(* PLC project CoDeSys External Library Template, WAGO e!COCKPIT e!COCKPIT, author 3S - Smart Software Solutions GmbH *)
(* stored: creationDateTime 2019-10-29T12:22:40.7625589, version 3.5.5.30, modificationDateTime 2019-10-24T14:40:07.960949, organization 3S - Smart Software Solutions GmbH *)
(* Library project template with all possible element types, docu and a sample project structure *)

FUNCTION_BLOCK fbUDPComm
  VAR_INPUT
    sIDSterownika : STRING;  (* ID sterownika *)
    sIDAplikacji : STRING;  (* ID aplikacji *)
    sMnemonik : STRING;  (* mnemonik właściciela *)
    sMACAdres : STRING;  (* MAC adres urządzenia - alias *)
    sMACAdresAplikacji : STRING;  (* MAC adres aplikacji - alias *)
    abMACAdresAplikacji : ARRAY[1..6] OF BYTE;  (* MAC adres aplikacji - wartość rzeczywista *)
    sDaneZapasowe : STRING;  (* dane zapasowe *)
    sAdresIP : STRING;  (* adres IP aplikacji *)
    wTransmitterPort : WORD;  (* port do wysyłania komunikatów *)
    wReceiverPort : WORD;  (* port nasłuchu *)
    sKluczSzyfrowania : STRING;
    intTablicaKomunikatowRozmiar : INT;
    intTablicaKomunikatowOverflow : INT;
    intTablicaKomunikatowZnacznikOdczytu : INT;
    iDetekcjaBlokadaKomunikacjiLimitIlosciRamek : INT;  (* Limit ilosi ramek do wysłania *)
    tDetekcjaBlokadaKomunikacjiLimitCzasu : TIME;
  END_VAR
  VAR_IN_OUT
    arTablicaKomunikatow : alARRAYTablicaKomunikatow;
    intTablicaKomunikatowZnacznikZapisu : INT;
    intTablicaKomunikatowZnacznikWysylkiUDP : INT;
    intTablicaKomunikatowLiczbaWBuforze : INT;
    intTransmitterLicznikKomunikatowWyslanych : INT;  (* zmienna zwierająca licznik komunikatów wysłanych pomiędzy heartbetami *)
    intReceiverLicznikKomunikatowOtrzymanych : INT;  (* zmienna zwierająca licznik komunikatów otrzymanych pomiędzy heartbetami *)
  END_VAR
  VAR
    fbTransmitter : fbBroadcaster;  (* definicja drivera wysyłającego broadcast pakietów UDP *)
    udiTransmitterNBytes : UDINT;  (* parametr drivera - ilość bajtów do wysłania *)
    xTransmitterClose : BOOL;  (* parametr drivera - zamknięcie portu komunikacyjnego *)
    xTransmitterTrigger : BOOL;  (* parametr drivera - uruchomienie wysłania telegramu *)
    sTransmitterTelegram : alSTRINGKomunikat;  (* zmienna zawierająca telegram do wysłania *)
    arTransmitterBuffer : ARRAY[1..512] OF BYTE;  (* tablica WORD bufora wysyłkowego *)
    pTransmitterBuffer : POINTER TO BYTE := ADR(arTransmitterBuffer[1]);  (* parametr drivera - pointer do tablicy bufora dla drivera wysyłającego *)
    fbReceiver : fbUdpReceiver;  (* definicja drivera odbierającego pakiety UDP *)
    xReceiverEnable : BOOL := TRUE;  (* parametr drivera - aktywacja działania drivera *)
    xReceiverOpen : BOOL := TRUE;  (* parametr drivera - otworzenie portu komunikacyjnego *)
    sReceiverTelegram : alSTRINGKomunikat;  (* zmienna zawierająca odebrany telegram *)
    arReceiverBuffer : ARRAY[1..512] OF BYTE;
    pReceiverBuffer : POINTER TO BYTE := ADR(arReceiverBuffer[1]);  (* parametr drivera - pointer do tablicy bufora dla drivera odbierającego *)
    intPetla : INT;  (* zmienna tymczasowa używana dla pętli *)
    arwHeartbeatTelegram : ARRAY[1..512] OF WORD;
    negUdpCommTxDone : F_TRIG;
    wCRC16_standard : WORD;
    intBlad : INT;
    sDane : alSTRINGKomunikat;
    sWyslanyKomunikat : alSTRINGKomunikat;
    typKomunikat : typKomunikat;
    xCRC16PakietOdebranyPoprawny : BOOL;
    arErrorKomunikat : ARRAY[0..20] OF alSTRINGKomunikat;  (* tablica przechowująca ostatni komunikat alarmu z danego kodu *)
    arErrorStan : ARRAY[1..20] OF BOOL;  (* tablica przechowująca stany alarmowe *)
    intTabelaKomunikatowZnacznikOdczytu : INT := 1;
    intEmergencyStopActiveZaraportowana : INT;
    sWyslanyKomunikatDummy : STRING;
    BlokadaKomunikacjiDetekcjaTriger : RS;  (* Blokada wysylania komunikatów *)
    BlokadaKomunikacjiDetekcjaTimer : TON;
    BlokadaKomunikacjiTriger : RS;
    fbBlokadaKomunikacjiTimer : TON;  (* Timer do cyklicznego wysyłania ramki z errorem blokady wysyłania ramek *)
    xBlokadaKomunikacji : BOOL;  (* Blokada komunikacji *)
    BlokadaKomunikacjiTimeDiff : TIME := TIME#200m0s0ms;
    xWyslijErrorBlokadyKomunikacji : BOOL;  (* Zmienna pomocniczna do fbWyslijErrorBlokadyKomunikacji *)
    fbWyslijErrorBlokadyKomunikacji : F_TRIG;  (* Zbocze opadające xWyslijErrorBlokadyKomunikacji *)
    xBlokadaKomunikacjiReset : BOOL;  (* Reset blokady komunikacji *)
    timestamp : STRING;  (* obsługa debugowania problemów z komunikatami *)
    dtCzasLokalny : DT;
    dtCzasKomunikatu : DT;
    tPrzesuniecie : TIME := TIME#5m0s0ms;
    xPrzekroczony : BOOL := FALSE;
    arTablicaBlednychKomunikatow : alARRAYTablicaKomunikatowDebug;
    uintZnacznikTablicyBlednychKomunikatow : UINT := 1;
    intTablicaKomunikatowZnacznikWysylkiUDP_Pamiec : INT := -1;
  END_VAR

            // jeśli wysyłanie telegramu zakończone OK wyczyść zmienną zawierającą telegram oraz wyzeruj licznik komunikatów wysłanych jeśli TO BYł heartbeat
// 2019-04-01 - JC Dodanie blokady wysylania komunikatów w przypadku przekroczenia limitu
// 2019-04-18 - AWy: Wysyłanie ramki z errorem blokady wysyłania ramek co minutę
// 2019-04-19 - AWy: Poprawienie mechanizmu resetu blokady i usunięcie tBlokadaKomunikacjiOpoznienie
// 2019-04-25 - AWy: Przeniesienie xBlokadaKomunikacjiReset z VAR_INPUT do VAR
// 2019-10-24 - AWy: Zmiana tPrzesuniecie na 300 sekund
IF NOT xTransmitterTrigger AND sTransmitterTelegram <> '' THEN
	IF fnKomunikatTyp(sTransmitterTelegram) = 'H' THEN
		intTransmitterLicznikKomunikatowWyslanych := 0;
	END_IF
	sTransmitterTelegram := '';
END_IF

IF sTransmitterTelegram = '' AND intTablicaKomunikatowZnacznikWysylkiUDP <> intTablicaKomunikatowZnacznikZapisu THEN
	fnTablicaKomunikatowInkrementacja(intWskaznik := intTablicaKomunikatowZnacznikWysylkiUDP , intRozmiarTablicy := intTablicaKomunikatowRozmiar);
	WHILE fnKomunikatMACAdres(arTablicaKomunikatow[intTablicaKomunikatowZnacznikWysylkiUDP]) <> sMACAdres AND intTablicaKomunikatowZnacznikWysylkiUDP <> intTablicaKomunikatowZnacznikZapisu DO
		fnTablicaKomunikatowInkrementacja(intWskaznik := intTablicaKomunikatowZnacznikWysylkiUDP , intRozmiarTablicy := intTablicaKomunikatowRozmiar);
 	END_WHILE
	IF fnKomunikatMACAdres(arTablicaKomunikatow[intTablicaKomunikatowZnacznikWysylkiUDP]) = sMACAdres THEN
		intTransmitterLicznikKomunikatowWyslanych := intTransmitterLicznikKomunikatowWyslanych + 1;
		//////////////////////////////////
		//Walidacja poprawności komunikatu
		//////////////////////////////////
		IF intTablicaKomunikatowZnacznikWysylkiUDP_Pamiec <> intTablicaKomunikatowZnacznikWysylkiUDP THEN
			timestamp := fnKomunikatSprawdzTimeStamp( sKomunikat:= arTablicaKomunikatow[intTablicaKomunikatowZnacznikWysylkiUDP],dtDataCzasWKomunikacie:=dtCzasKomunikatu, dtDataCzasAktualny:=dtCzasLokalny);
			IF(dtCzasKomunikatu + tPrzesuniecie) < dtCzasLokalny THEN
				xPrzekroczony := TRUE;
				arTablicaBlednychKomunikatow[uintZnacznikTablicyBlednychKomunikatow].dtLokalnyCzasSterownika := dtCzasLokalny;
				arTablicaBlednychKomunikatow[uintZnacznikTablicyBlednychKomunikatow].intGlobalnaLiczbaKomunikatowWBuforze := intTablicaKomunikatowLiczbaWBuforze;
				arTablicaBlednychKomunikatow[uintZnacznikTablicyBlednychKomunikatow].intGlobalnyZnacznikOdczytu := intTablicaKomunikatowZnacznikOdczytu;
				arTablicaBlednychKomunikatow[uintZnacznikTablicyBlednychKomunikatow].intGlobalnyZnacznikWysylkiUDP := intTablicaKomunikatowZnacznikWysylkiUDP;
				arTablicaBlednychKomunikatow[uintZnacznikTablicyBlednychKomunikatow].intGlobalnyZnacznikZapisu := intTablicaKomunikatowZnacznikZapisu;
				arTablicaBlednychKomunikatow[uintZnacznikTablicyBlednychKomunikatow].sDane := arTablicaKomunikatow[intTablicaKomunikatowZnacznikWysylkiUDP];
				IF uintZnacznikTablicyBlednychKomunikatow < 99 THEN
					uintZnacznikTablicyBlednychKomunikatow := uintZnacznikTablicyBlednychKomunikatow + 1;
				ELSE
					uintZnacznikTablicyBlednychKomunikatow := 1;
				END_IF
				//skasuj atrybuty
				arTablicaKomunikatow[intTablicaKomunikatowZnacznikWysylkiUDP] := MID(arTablicaKomunikatow[intTablicaKomunikatowZnacznikWysylkiUDP], 82, 1);
				arTablicaKomunikatow[intTablicaKomunikatowZnacznikWysylkiUDP] := CONCAT(arTablicaKomunikatow[intTablicaKomunikatowZnacznikWysylkiUDP], 'BLADRAMKI=2');
			ELSE
				xPrzekroczony := FALSE;
			END_IF
			intTablicaKomunikatowZnacznikWysylkiUDP_Pamiec := intTablicaKomunikatowZnacznikWysylkiUDP;
		END_IF
		//////////////////////////////////
		fnAES256Szyfrowanie(	sKomunikat := arTablicaKomunikatow[intTablicaKomunikatowZnacznikWysylkiUDP] , 
								sKlucz := sKluczSzyfrowania , 
								intError := intBlad , 
								sKomunikatZaszyfrowany := sTransmitterTelegram);
		
		fnCRC16Wysylanie(	sKomunikat :=  sTransmitterTelegram,
							arTransmitterBuffer := arTransmitterBuffer ,
							udiTransmitterNBytes := udiTransmitterNBytes);
		xTransmitterTrigger := TRUE;
	END_IF
END_IF

// driver wysyłający pakiety UDP

// Blokada wysyłania komunikatów - po przekroczeniu iDetekcjaBlokadaKomunikacjiLimitIlosciRamek w czasie tDetekcjaBlokadaKomunikacjiLimitCzasu algorytm zatrzyma wysyłanie ramek, ale nie 
// przestanie zapisywać ich do tablicy. Raz na minutę zostanie wysłana ramka E informująca o blokadzie. Funkcjonalność ma na celu zabezpieczenia systemu przed spamowaniem ramkami jako 
// konsekwencji błędów programistycznych. 

BlokadaKomunikacjiDetekcjaTriger(Set := (intTablicaKomunikatowZnacznikZapisu = (intTablicaKomunikatowRozmiar - iDetekcjaBlokadaKomunikacjiLimitIlosciRamek)),
								 RESET1 := (intTablicaKomunikatowZnacznikZapisu = intTablicaKomunikatowRozmiar)); // Sprawdzenie następuje, gdy znacznik jest w połowie tablicy komunikatów
IF BlokadaKomunikacjiDetekcjaTimer.ET <> T#0MS AND BlokadaKomunikacjiDetekcjaTriger.RESET1 = TRUE AND NOT xBlokadaKomunikacjiReset THEN
	BlokadaKomunikacjiTimeDiff := BlokadaKomunikacjiDetekcjaTimer.ET; 
END_IF

IF xBlokadaKomunikacjiReset THEN
	BlokadaKomunikacjiTimeDiff := T#200M;
END_IF

BlokadaKomunikacjiDetekcjaTimer(IN := BlokadaKomunikacjiDetekcjaTriger.Q1, PT := T#100S);
 
BlokadaKomunikacjiTriger(Set := (BlokadaKomunikacjiTimeDiff < tDetekcjaBlokadaKomunikacjiLimitCzasu), RESET1 := xBlokadaKomunikacjiReset, Q1 => xBlokadaKomunikacji); 

IF NOT(xBlokadaKomunikacji) THEN
	udiTransmitterNBytes := INT_TO_UDINT(LEN(sTransmitterTelegram)) + 2;
	fbTransmitter(	sNetName := sAdresIP ,
					wPort := wTransmitterPort , 
					pTxBuffer := pTransmitterBuffer , 
					udiTxNBytes := udiTransmitterNBytes , 
					xClose := xTransmitterClose , 
					xTxTrigger := xTransmitterTrigger);
END_IF

// driver nasłuchujący pakietów UDP

fbReceiver(	wPort := wReceiverPort , 
			pRxBuffer := pReceiverBuffer , 
			udiRxBufferSize := 512 , 
			xRxEnable := xReceiverEnable , 
			xOpen := xReceiverOpen);

// po otrzymaniu pakietu wykonanie zapisu danych kontroli CRC itd

IF fbReceiver.xPacketReceived = TRUE THEN
	sReceiverTelegram := LEFT(sReceiverTelegram , UDINT_TO_INT(fbReceiver.udiRxNBytes));
	fnAES256Odszyfrowanie(	sKomunikatZaszyfrowany := sReceiverTelegram , 
							sKlucz := sKluczSzyfrowania ,
							intError := intBlad ,
							sKomunikat := sReceiverTelegram);

// sprawdzenie CRC otrzymanego komunikatu

	xCRC16PakietOdebranyPoprawny := fnCRC16Odbieranie(	arReceiverBuffer := arReceiverBuffer ,
														udiRxNBytes := fbReceiver.udiRxNBytes ,
														sMACAdresAplikacji := sMACAdresAplikacji ,
														abMACAdresAplikacji := abMACAdresAplikacji ,
														sKomunikat := sReceiverTelegram);
	IF xCRC16PakietOdebranyPoprawny THEN

// CRC poprawne zapis komunikatu do tablicy komunikatów otrzymanych o nie jest to komunikat z tego sterownika

		intReceiverLicznikKomunikatowOtrzymanych := intReceiverLicznikKomunikatowOtrzymanych + 1;

		IF fnKomunikatMACAdres(sReceiverTelegram) <> sMACAdres THEN
			fnZapiszKomunikat(	sCalyKomunikat := sReceiverTelegram ,
								sTypKomunikatu := '' ,
								sMnemonik := '' ,
								sMACAdres := '' ,
								sIDNadawcy := '' ,
								sIDOdbiorcy := '' ,
								sDaneZapasowe := '' ,
								sDane := '' ,
								arTablicaKomunikatow := arTablicaKomunikatow ,
								intTablicaKomunikatowZnacznikZapisu := intTablicaKomunikatowZnacznikZapisu ,
								intTablicaKomunikatowRozmiar := intTablicaKomunikatowRozmiar ,
								sWyslanyKomunikat := sWyslanyKomunikat);
		END_IF
		
// sprawdzenie statusu błędu jeśli błąd był zaraportowany zaraportowanie poprawnego CRC

		IF arErrorStan[enumSystemErrorKlasa.BladCRCWKomunikacieZIZE] THEN
			arErrorStan[enumSystemErrorKlasa.BladCRCWKomunikacieZIZE] := FALSE;
			sDane := CONCAT('ACT=0;CLASS=' , INT_TO_STRING(enumSystemErrorKlasa.BladCRCWKomunikacieZIZE));
			sDane := CONCAT(sDane , ';NUM=');
			sDane := CONCAT(sDane , INT_TO_STRING(enumSystemError.BladCRCWKomunikacieZIZE));
			sDane := CONCAT(sDane , ';E');
			sDane := CONCAT(sDane , fnKonwersjaINT_STRING(intWartosc := enumSystemError.BladCRCWKomunikacieZIZE , intIloscZnakow := 3));
			sDane := CONCAT(sDane , 'ACT=0');
			fnZapiszKomunikat(	sCalyKomunikat := '' ,
								sTypKomunikatu := 'E' ,
								sMnemonik :=  sMnemonik ,
								sMACAdres := sMACAdres ,
								sIDNadawcy := sIdSterownika ,
								sIDOdbiorcy := sIdAplikacji ,
								sDaneZapasowe := sDaneZapasowe ,
								sDane := sDane ,
								arTablicaKomunikatow := arTablicaKomunikatow ,
								intTablicaKomunikatowZnacznikZapisu := intTablicaKomunikatowZnacznikZapisu ,
								intTablicaKomunikatowRozmiar := intTablicaKomunikatowRozmiar ,
								sWyslanyKomunikat := arErrorKomunikat[enumSystemError.BladCRCWKomunikacieZIZE]);
			END_IF
		ELSE

// jeżeli był błąd w CRC komunikatu i poprzednie komunikaty były bez błędu zaraportuj ten błąd z powrotem do IZE

		IF NOT arErrorStan[enumSystemErrorKlasa.BladCRCWKomunikacieZIZE] THEN
			arErrorStan[enumSystemErrorKlasa.BladCRCWKomunikacieZIZE] := TRUE;
			sDane := CONCAT('ACT=1;CLASS=' , INT_TO_STRING(enumSystemErrorKlasa.BladCRCWKomunikacieZIZE));
			sDane := CONCAT(sDane , ';NUM=');
			sDane := CONCAT(sDane , INT_TO_STRING(enumSystemError.BladCRCWKomunikacieZIZE));	
			sDane := CONCAT(sDane , ';E');
			sDane := CONCAT(sDane , fnKonwersjaINT_STRING(intWartosc := enumSystemError.BladCRCWKomunikacieZIZE , intIloscZnakow := 3));
			sDane := CONCAT(sDane , 'ACT=1');
			fnZapiszKomunikat(	sCalyKomunikat := '' ,
								sTypKomunikatu := 'E' ,
								sMnemonik :=  sMnemonik,
								sMACAdres := sMACAdres ,
								sIDNadawcy := sIdSterownika ,
								sIDOdbiorcy := sIdAplikacji ,
								sDaneZapasowe := sDaneZapasowe ,
								sDane := sDane ,
								arTablicaKomunikatow := arTablicaKomunikatow ,
								intTablicaKomunikatowZnacznikZapisu := intTablicaKomunikatowZnacznikZapisu ,
								intTablicaKomunikatowRozmiar := intTablicaKomunikatowRozmiar ,
								sWyslanyKomunikat := arErrorKomunikat[enumSystemError.BladCRCWKomunikacieZIZE]);
		END_IF
	END_IF
END_IF

// obsługa alarmu przepełnienia bufora komunikatów

intTablicaKomunikatowLiczbaWBuforze := intTablicaKomunikatowZnacznikZapisu - intTablicaKomunikatowZnacznikWysylkiUDP;

IF intTablicaKomunikatowLiczbaWBuforze < 0 THEN
	intTablicaKomunikatowLiczbaWBuforze := intTablicaKomunikatowLiczbaWBuforze + intTablicaKomunikatowRozmiar;
END_IF

IF intTablicaKomunikatowLiczbaWBuforze > intTablicaKomunikatowOverflow AND NOT arErrorStan[enumSystemError.ZaDuzaIloscKomunikatowWBuforze] THEN
	arErrorStan[enumSystemError.ZaDuzaIloscKomunikatowWBuforze] := TRUE;
	sDane := CONCAT('ACT=1;CLASS=' , INT_TO_STRING(enumSystemErrorKlasa.ZaDuzaIloscKomunikatowWBuforze));
	sDane := CONCAT(sDane , ';NUM=');
	sDane := CONCAT(sDane , INT_TO_STRING(enumSystemError.ZaDuzaIloscKomunikatowWBuforze));	
	sDane := CONCAT(sDane , ';E');
	sDane := CONCAT(sDane , fnKonwersjaINT_STRING(intWartosc := enumSystemError.ZaDuzaIloscKomunikatowWBuforze , intIloscZnakow := 3));
	sDane := CONCAT(sDane , 'ACT=1');
	fnZapiszKomunikat(	sCalyKomunikat := '' ,
						sTypKomunikatu := 'E' ,
						sMnemonik :=  sMnemonik ,
						sMACAdres := sMACAdres ,
						sIDNadawcy := sIdSterownika ,
						sIDOdbiorcy := sIdAplikacji ,
						sDaneZapasowe := sDaneZapasowe ,
						sDane := sDane ,
						arTablicaKomunikatow := arTablicaKomunikatow ,
						intTablicaKomunikatowZnacznikZapisu := intTablicaKomunikatowZnacznikZapisu ,
						intTablicaKomunikatowRozmiar := intTablicaKomunikatowRozmiar ,
						sWyslanyKomunikat := arErrorKomunikat[enumSystemError.ZaDuzaIloscKomunikatowWBuforze]);						
END_IF
IF  intTablicaKomunikatowLiczbaWBuforze = 0 AND arErrorStan[enumSystemError.ZaDuzaIloscKomunikatowWBuforze] THEN
	arErrorStan[enumSystemError.ZaDuzaIloscKomunikatowWBuforze] := FALSE;
	sDane := CONCAT('ACT=0;CLASS=' , INT_TO_STRING(enumSystemErrorKlasa.ZaDuzaIloscKomunikatowWBuforze));
	sDane := CONCAT(sDane , ';NUM=');
	sDane := CONCAT(sDane , INT_TO_STRING(enumSystemError.ZaDuzaIloscKomunikatowWBuforze));	
	sDane := CONCAT(sDane , ';E');
	sDane := CONCAT(sDane , fnKonwersjaINT_STRING(intWartosc := enumSystemError.ZaDuzaIloscKomunikatowWBuforze , intIloscZnakow := 3));
	sDane := CONCAT(sDane , 'ACT=0');
	fnZapiszKomunikat(	sCalyKomunikat := '' ,
						sTypKomunikatu := 'E' ,
						sMnemonik :=  sMnemonik,
						sMACAdres := sMACAdres ,
						sIDNadawcy := sIdSterownika ,
						sIDOdbiorcy := sIdAplikacji ,
						sDaneZapasowe := sDaneZapasowe ,
						sDane := sDane ,
						arTablicaKomunikatow := arTablicaKomunikatow ,
						intTablicaKomunikatowZnacznikZapisu := intTablicaKomunikatowZnacznikZapisu ,
						intTablicaKomunikatowRozmiar := intTablicaKomunikatowRozmiar ,
						sWyslanyKomunikat := arErrorKomunikat[enumSystemError.ZaDuzaIloscKomunikatowWBuforze]);
END_IF


// obsługa alarmu - blokada wysyłania komunikatów ze względu na za dużą ilość wysyłanych ramek (wysyłanie ramki co 1 minutę)

IF xBlokadaKomunikacji THEN
	arErrorStan[enumSystemError.BlokadaWysylaniaRamek] := TRUE;
	fbBlokadaKomunikacjiTimer(IN := xWyslijErrorBlokadyKomunikacji, PT := T#1M);
	xWyslijErrorBlokadyKomunikacji := TRUE;
	IF fbBlokadaKomunikacjiTimer.Q  THEN														// Wyślij error zaraz co 1 minutę
		xWyslijErrorBlokadyKomunikacji := FALSE;
		intTablicaKomunikatowZnacznikWysylkiUDP := intTablicaKomunikatowZnacznikZapisu;			// Ustaw znacznik wysyłania na aktualnie zapisywanej ramce
		// Sklejenie ramki z komunikatem o błędzie
		sDane := CONCAT('ACT=1;CLASS=' , INT_TO_STRING(enumSystemErrorKlasa.BlokadaWysylaniaRamek));
		sDane := CONCAT(sDane , ';NUM=');
		sDane := CONCAT(sDane , INT_TO_STRING(enumSystemError.BlokadaWysylaniaRamek));	
		sDane := CONCAT(sDane , ';E');
		sDane := CONCAT(sDane , fnKonwersjaINT_STRING(intWartosc := enumSystemError.BlokadaWysylaniaRamek , intIloscZnakow := 3));
		sDane := CONCAT(sDane , 'ACT=1');
		fnZapiszKomunikat(	sCalyKomunikat := '' ,
							sTypKomunikatu := 'E' ,
							sMnemonik :=  sMnemonik ,
							sMACAdres := sMACAdres ,
							sIDNadawcy := sIdSterownika ,
							sIDOdbiorcy := sIdAplikacji ,
							sDaneZapasowe := sDaneZapasowe ,
							sDane := sDane ,
							arTablicaKomunikatow := arTablicaKomunikatow ,
							intTablicaKomunikatowZnacznikZapisu := intTablicaKomunikatowZnacznikZapisu ,
							intTablicaKomunikatowRozmiar := intTablicaKomunikatowRozmiar ,
							sWyslanyKomunikat := arErrorKomunikat[enumSystemError.BlokadaWysylaniaRamek]);
		sTransmitterTelegram := arErrorKomunikat[enumSystemError.BlokadaWysylaniaRamek];	
	END_IF
	fbWyslijErrorBlokadyKomunikacji(CLK := xWyslijErrorBlokadyKomunikacji);
	IF fbWyslijErrorBlokadyKomunikacji.Q THEN
		// Wysłanie ramki		
		fnCRC16Wysylanie(	sKomunikat :=  sTransmitterTelegram,
							arTransmitterBuffer := arTransmitterBuffer ,
							udiTransmitterNBytes := udiTransmitterNBytes);				
		udiTransmitterNBytes := INT_TO_UDINT(LEN(sTransmitterTelegram)) + 2;
		fbTransmitter(	sNetName := sAdresIP ,
						wPort := wTransmitterPort , 
						pTxBuffer := pTransmitterBuffer , 
						udiTxNBytes := udiTransmitterNBytes , 
						xClose := xTransmitterClose , 
						xTxTrigger := xTransmitterTrigger);
	END_IF
END_IF
IF  NOT (BlokadaKomunikacjiTriger.Q1) AND arErrorStan[enumSystemError.BlokadaWysylaniaRamek] THEN
	arErrorStan[enumSystemError.BlokadaWysylaniaRamek] := FALSE;
	sDane := CONCAT('ACT=0;CLASS=' , INT_TO_STRING(enumSystemErrorKlasa.BlokadaWysylaniaRamek));
	sDane := CONCAT(sDane , ';NUM=');
	sDane := CONCAT(sDane , INT_TO_STRING(enumSystemError.BlokadaWysylaniaRamek));	
	sDane := CONCAT(sDane , ';E');
	sDane := CONCAT(sDane , fnKonwersjaINT_STRING(intWartosc := enumSystemError.BlokadaWysylaniaRamek , intIloscZnakow := 3));
	sDane := CONCAT(sDane , 'ACT=0');
	fnZapiszKomunikat(	sCalyKomunikat := '' ,
						sTypKomunikatu := 'E' ,
						sMnemonik :=  sMnemonik,
						sMACAdres := sMACAdres ,
						sIDNadawcy := sIdSterownika ,
						sIDOdbiorcy := sIdAplikacji ,
						sDaneZapasowe := sDaneZapasowe ,
						sDane := sDane ,
						arTablicaKomunikatow := arTablicaKomunikatow ,
						intTablicaKomunikatowZnacznikZapisu := intTablicaKomunikatowZnacznikZapisu ,
						intTablicaKomunikatowRozmiar := intTablicaKomunikatowRozmiar ,
						sWyslanyKomunikat := arErrorKomunikat[enumSystemError.BlokadaWysylaniaRamek]);
END_IF


//????????
IF intTabelaKomunikatowZnacznikOdczytu <> intTablicaKomunikatowZnacznikZapisu THEN
	fnTablicaKomunikatowInkrementacja(intRozmiarTablicy := intTablicaKomunikatowRozmiar , intWskaznik := intTabelaKomunikatowZnacznikOdczytu);
	IF fnIDOdbiorcyMatch(arTablicaKomunikatow[intTabelaKomunikatowZnacznikOdczytu] , sIDSterownika) THEN
		IF fnKomunikatTyp(arTablicaKomunikatow[intTabelaKomunikatowZnacznikOdczytu]) = 'Q' THEN
//			IF fnKomunikatDaneSzukajZmiennej(arTablicaKomunikatow[intTabelaKomunikatowZnacznikOdczytu] , 'ALARM') OR 
//				fnKomunikatDaneSzukajZmiennej(arTablicaKomunikatow[intTabelaKomunikatowZnacznikOdczytu] , 'ALL') THEN
//				FOR intPetla := 1 TO 20 BY 1 DO
//					IF arErrorKomunikat[intPetla] <> '' THEN
//						fnZapiszKomunikat(	sCalyKomunikat := arErrorKomunikat[intPetla] ,
//											sTypKomunikatu := '' ,
//											sMnemonik := '' ,
//											sMACAdres := '' ,
//											sIDNadawcy := '' ,
//											sIDOdbiorcy := '' ,
//											sDaneZapasowe := '' ,
//											sDane := '' ,
//											arTablicaKomunikatow := arTablicaKomunikatow ,
//											intTablicaKomunikatowZnacznikZapisu := intTablicaKomunikatowZnacznikZapisu ,
//											intTablicaKomunikatowRozmiar := intTablicaKomunikatowRozmiar ,
//											sWyslanyKomunikat := sWyslanyKomunikat);
//					END_IF
//				END_FOR
//			END_IF	
///wrzucic nowy Q
		END_IF
	END_IF
END_IF
          
END_FUNCTION_BLOCK
